Fanuc TP program (LS listing): GRIPPER1.LS

/PROG  GRIPPER1	  Macro
/ATTR
OWNER		= MNEDITOR;
COMMENT		= "";
PROG_SIZE	= 237;
CREATE		= DATE 25-02-04  TIME 18:17:10;
MODIFIED	= DATE 25-02-04  TIME 18:20:22;
FILE_NAME	= ;
VERSION		= 0;
LINE_COUNT	= 5;
MEMORY_SIZE	= 589;
PROTECT		= READ_WRITE;
TCD:  STACK_SIZE	= 0,
      TASK_PRIORITY	= 50,
      TIME_SLICE	= 0,
      BUSY_LAMP_OFF	= 0,
      ABORT_REQUEST	= 0,
      PAUSE_REQUEST	= 0;
DEFAULT_GROUP	= *,*,*,*,*;
CONTROL_CODE	= 00000000 00000000;
LOCAL_REGISTERS	= 0,0,0;
/APPL

AUTO_SINGULARITY_HEADER;
  ENABLE_SINGULARITY_AVOIDANCE   : TRUE;
/MN
   1:  IF (RO[1]=OFF) THEN ;
   2:  RO[1]=ON ;
   3:  ELSE ;
   4:  RO[1]=OFF ;
   5:  ENDIF ;
/POS
/END
